Staubli VAL3: setEventAndWait.pgx

public program setEventAndWait(num handle_, num event_, bool& result_[])
begin
  // set event and wait for processing
  nCommand[handle_]=coSW
  call sendCommand(handle_,"sw"+toString("0.0",event_),result_)
end
